PROGRAM Main
VAR
	// Motors
	{attribute 'TcLinkTo' := '.bLimitForwardEnable:=TIIB[VonHamos_EL7041_E1]^STM Status^Status^Digital input 1;
                              .bLimitBackwardEnable:=TIIB[VonHamos_EL7041_E1]^STM Status^Status^Digital input 2'}
	{attribute 'pytmc' := '
		pv: HXX:VON_HAMOS:MMS:01
	'}
	M1 : DUT_MotionStage; // Y axis

	fbMotionStageM1 : FB_MotionStage;
END_VAR

// Hardware Enable
M1.bHardwareEnable := TRUE;
fbMotionStageM1(stMotionStage:=M1);

END_PROGRAM

(* stored: Version 1.1.0.1, ProductVersion 3.1.4022.18
   POU Main: Id {90ca38b8-fcf5-47a7-9a91-8e230c16c364}, SpecialFunc None *)
